FUNCTION_BLOCK EQUIP_Sorter (* Composite Function Block Type *)
  (* Standard: 61499-2 *)
  (* Version 0.0, 08/01/2026, Schneider Electric, template *)
  PACKAGE Main;
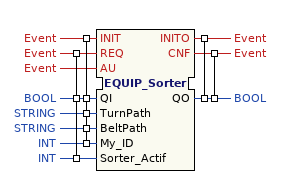
  EVENT_INPUT
    INIT WITH QI, TurnPath, BeltPath, My_ID; (* Initialization Request *)
    REQ WITH QI, Sorter_Actif; (* Normal Execution Request *)
    AU; (* Arret urgence *)
  END_EVENT
  EVENT_OUTPUT
    INITO WITH QO; (* Initialization Confirm *)
    CNF WITH QO; (* Execution Confirmation *)
  END_EVENT
  VAR_INPUT
    QI : BOOL; (* Input event qualifier *)
    TurnPath : STRING;
    BeltPath : STRING;
    My_ID : INT;
    Sorter_Actif : INT;
  END_VAR
  VAR_OUTPUT
    QO : BOOL; (* Output event qualifier *)
  END_VAR
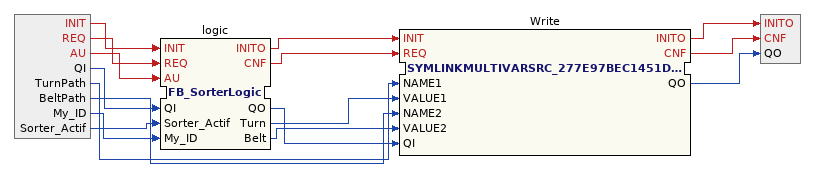
  FBS
    logic : FB_SorterLogic;
    Write : SYMLINKMULTIVARSRC_277E97BEC1451D2C; {SET_ATTRIBUTE(Configuration.GenericFBType.InterfaceParams, Runtime.System#I:=2;VALUE${I$}:BOOL,BOOL)}
  END_FBS
  EVENT_CONNECTIONS
    INIT TO logic.INIT;
    REQ TO logic.REQ;
    AU TO logic.AU;
    logic.INITO TO Write.INIT;
    logic.CNF TO Write.REQ;
    Write.INITO TO INITO;
    Write.CNF TO CNF;
  END_CONNECTIONS
  DATA_CONNECTIONS
    QI TO logic.QI;
    TurnPath TO Write.NAME1;
    logic.Turn TO Write.VALUE1;
    BeltPath TO Write.NAME2;
    logic.Belt TO Write.VALUE2;
    Write.QO TO QO;
    Sorter_Actif TO logic.Sorter_Actif;
    My_ID TO logic.My_ID;
    logic.QO TO Write.QI;
  END_CONNECTIONS
END_FUNCTION_BLOCK
